// SIMATIC STEP 7 (V5.x) project T 13  27
// program: Programa S7(1)

SYMBOL_TABLE
"FLANCOS"	DB 1	DB 1
"PMARCHA"	I 0.0	BOOL
"PPARO"	I 0.1	BOOL
"Cycle Execution"	OB 1	OB 1
"MOTOR"	Q 0.0	BOOL
END_SYMBOL_TABLE
